// TIA Portal V20 export
VAR_GLOBAL   // PLC tag table "LPMLV2022_Constants"
END_VAR
VAR_GLOBAL CONSTANT   // user constants
   LPMLV2022_MODE_INVALID : DInt := 0;   // OMAC PackMLV2022 unit mode Invalid
   LPMLV2022_MODE_PRODUCTION : DInt := 1;   // OMAC PackMLV2022 unit mode Production
   LPMLV2022_MODE_MAINTENANCE : DInt := 2;   // OMAC PackMLV2022 unit mode Maintenance
   LPMLV2022_MODE_MANUAL : DInt := 3;   // OMAC PackMLV2022 unit mode Manual
   LPMLV2022_MODE_USER_01 : DInt := 4;   // OMAC PackMLV2022 user-defined unit mode 01
   LPMLV2022_MODE_USER_02 : DInt := 5;   // OMAC PackMLV2022 user-defined unit mode 02
   LPMLV2022_MODE_USER_03 : DInt := 6;   // OMAC PackMLV2022 user-defined unit mode 03
   LPMLV2022_MODE_USER_04 : DInt := 7;   // OMAC PackMLV2022 user-defined unit mode 04
   LPMLV2022_MODE_USER_05 : DInt := 8;   // OMAC PackMLV2022 user-defined unit mode 05
   LPMLV2022_MODE_USER_06 : DInt := 9;   // OMAC PackMLV2022 user-defined unit mode 06
   LPMLV2022_MODE_USER_07 : DInt := 10;   // OMAC PackMLV2022 user-defined unit mode 07
   LPMLV2022_MODE_USER_08 : DInt := 11;   // OMAC PackMLV2022 user-defined unit mode 08
   LPMLV2022_MODE_USER_09 : DInt := 12;   // OMAC PackMLV2022 user-defined unit mode 09
   LPMLV2022_MODE_USER_10 : DInt := 13;   // OMAC PackMLV2022 user-defined unit mode 10
   LPMLV2022_MODE_USER_11 : DInt := 14;   // OMAC PackMLV2022 user-defined unit mode 11
   LPMLV2022_MODE_USER_12 : DInt := 15;   // OMAC PackMLV2022 user-defined unit mode 12
   LPMLV2022_MODE_USER_13 : DInt := 16;   // OMAC PackMLV2022 user-defined unit mode 13
   LPMLV2022_MODE_USER_14 : DInt := 17;   // OMAC PackMLV2022 user-defined unit mode 14
   LPMLV2022_MODE_USER_15 : DInt := 18;   // OMAC PackMLV2022 user-defined unit mode 15
   LPMLV2022_MODE_USER_16 : DInt := 19;   // OMAC PackMLV2022 user-defined unit mode 16
   LPMLV2022_MODE_USER_17 : DInt := 20;   // OMAC PackMLV2022 user-defined unit mode 17
   LPMLV2022_MODE_USER_18 : DInt := 21;   // OMAC PackMLV2022 user-defined unit mode 18
   LPMLV2022_MODE_USER_19 : DInt := 22;   // OMAC PackMLV2022 user-defined unit mode 19
   LPMLV2022_MODE_USER_20 : DInt := 23;   // OMAC PackMLV2022 user-defined unit mode 20
   LPMLV2022_MODE_USER_21 : DInt := 24;   // OMAC PackMLV2022 user-defined unit mode 21
   LPMLV2022_MODE_USER_22 : DInt := 25;   // OMAC PackMLV2022 user-defined unit mode 22
   LPMLV2022_MODE_USER_23 : DInt := 26;   // OMAC PackMLV2022 user-defined unit mode 23
   LPMLV2022_MODE_USER_24 : DInt := 27;   // OMAC PackMLV2022 user-defined unit mode 24
   LPMLV2022_MODE_USER_25 : DInt := 28;   // OMAC PackMLV2022 user-defined unit mode 25
   LPMLV2022_MODE_USER_26 : DInt := 29;   // OMAC PackMLV2022 user-defined unit mode 26
   LPMLV2022_MODE_USER_27 : DInt := 30;   // OMAC PackMLV2022 user-defined unit mode 27
   LPMLV2022_MODE_USER_28 : DInt := 31;   // OMAC PackMLV2022 user-defined unit mode 28
   LPMLV2022_STATE_UNDEFINED : DInt := 0;   // OMAC PackMLV2022 state Undefined
   LPMLV2022_STATE_CLEARING : DInt := 1;   // OMAC PackMLV2022 state Clearing
   LPMLV2022_STATE_STOPPED : DInt := 2;   // OMAC PackMLV2022 state Stopped
   LPMLV2022_STATE_STARTING : DInt := 3;   // OMAC PackMLV2022 state Starting
   LPMLV2022_STATE_IDLE : DInt := 4;   // OMAC PackMLV2022 state Idle
   LPMLV2022_STATE_SUSPENDED : DInt := 5;   // OMAC PackMLV2022 state Suspended
   LPMLV2022_STATE_EXECUTE : DInt := 6;   // OMAC PackMLV2022 state Execute
   LPMLV2022_STATE_STOPPING : DInt := 7;   // OMAC PackMLV2022 state Stopping
   LPMLV2022_STATE_ABORTING : DInt := 8;   // OMAC PackMLV2022 state Aborting
   LPMLV2022_STATE_ABORTED : DInt := 9;   // OMAC PackMLV2022 state Aborted
   LPMLV2022_STATE_HOLDING : DInt := 10;   // OMAC PackMLV2022 state Holding
   LPMLV2022_STATE_HELD : DInt := 11;   // OMAC PackMLV2022 state Held
   LPMLV2022_STATE_UNHOLDING : DInt := 12;   // OMAC PackMLV2022 state Unholding
   LPMLV2022_STATE_SUSPENDING : DInt := 13;   // OMAC PackMLV2022 state Suspending
   LPMLV2022_STATE_UNSUSPENDING : DInt := 14;   // OMAC PackMLV2022 state Unsuspending
   LPMLV2022_STATE_RESETTING : DInt := 15;   // OMAC PackMLV2022 state Resetting
   LPMLV2022_STATE_COMPLETING : DInt := 16;   // OMAC PackMLV2022 state Completing
   LPMLV2022_STATE_COMPLETED : DInt := 17;   // OMAC PackMLV2022 state Completed
   LPMLV2022_CMD_UNDEFINED : DInt := 0;   // OMAC PackMLV2022 control command Undefined
   LPMLV2022_CMD_RESET : DInt := 1;   // OMAC PackMLV2022 control command Reset
   LPMLV2022_CMD_START : DInt := 2;   // OMAC PackMLV2022 control command Start
   LPMLV2022_CMD_STOP : DInt := 3;   // OMAC PackMLV2022 control command Stop
   LPMLV2022_CMD_HOLD : DInt := 4;   // OMAC PackMLV2022 control command Hold
   LPMLV2022_CMD_UNHOLD : DInt := 5;   // OMAC PackMLV2022 control command Unhold
   LPMLV2022_CMD_SUSPEND : DInt := 6;   // OMAC PackMLV2022 control command Suspend
   LPMLV2022_CMD_UNSUSPEND : DInt := 7;   // OMAC PackMLV2022 control command Unsuspend
   LPMLV2022_CMD_ABORT : DInt := 8;   // OMAC PackMLV2022 control command Abort
   LPMLV2022_CMD_CLEAR : DInt := 9;   // OMAC PackMLV2022 control command Clear
   LPMLV2022_CMD_COMPLETE : DInt := 10;   // OMAC PackMLV2022 control command Complete
   LPMLV2022_DIAG_BUFFER_UPPER_LIM : Int := 7;   // Diagnostics buffer array upper boundary (0-based)
   LPMLV2022_STATES_UPPER_LIM : Int := 17;   // (Number of states - 1) -> Array[0..LPMLV2022_STATES_UPPER_LIM]
   LPMLV2022_MAX_MODES_UPPER_LIM : Int := 16;   // (Maximum number of unit modes - 1) -> Array[0..LPMLV2022_MAX_MODES_UPPER_LIM]
   LPMLV2022_MODES_UPPER_LIM : Int := 16;   // (Number of unit modes - 1) -> Array[0..LPMLV2022_MODES_UPPER_LIM]
END_VAR
